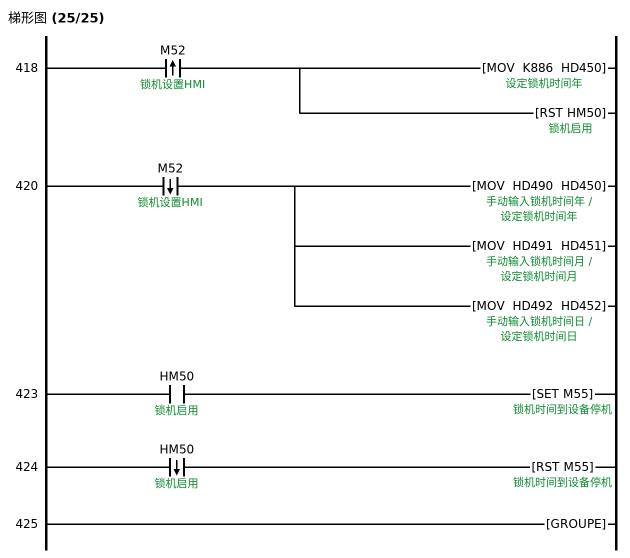
[picture p24: 梯形图 rows 418-425]
LDP    M52	; 锁机设置HMI
MOV    K886 HD450	; 设定锁机时间年
RST    HM50	; 锁机启用
LDF    M52	; 锁机设置HMI
MOV    HD490 HD450	; 手动输入锁机时间年 / 设定锁机时间年
MOV    HD491 HD451	; 手动输入锁机时间月 / 设定锁机时间月
MOV    HD492 HD452	; 手动输入锁机时间日 / 设定锁机时间日
LD     HM50	; 锁机启用
SET    M55	; 锁机时间到设备停机
LDF    HM50	; 锁机启用
RST    M55	; 锁机时间到设备停机
GROUPE

COMMENTS (devices not used above)
M3	急停HMI
M5	NG清料HMI
M6	轴复位HMI
M8	参数默认HMI
M9	产量清零HMI
M10	当前产量清零HMI
M21	軸总復位中
M22	设备复位中
M25	设备清料完成
M2042	轴2_JOG快慢速HMI
M2021	轴1_JOG- HMI
M2022	轴2_JOG- HMI
M2041	轴1_JOG快慢速HMI
M2002	轴2_JOG+ HMI
M1821	与读码器通信异常
D2100	轴1_JOG快速度
D2102	轴1_JOG慢速度
D2104	轴1_JOG速度寄存
D2106	轴1_JOG增量
D2108	轴1_JOG位置寄存
D2110	轴1_回零速度
D2112	轴1_运行速度
D2114	轴1_自动加速度
D2115	轴1_自动减速度
D2116	轴1_JOG加速度
D2117	轴1_JOG减速度
D2118	轴1_定位位置寄存
M2141	轴1_伺服回零中
M1200	快慢速切换HMI
M1020	从1#Y0 左侧三色灯（红）       HMI
HD8	切鼻梁个数计数
HD12	滚刀切料个数计数
M2001	轴1_JOG+ HMI
HD40	Y0当前脉冲值记忆
HD42	Y1当前脉冲值记忆
T2	超声波休眠延时
HD2	超声波休眠时间
T3	超声运行延时
D110	从5读码寄存
D112	从6读码寄存
D114	从7读码寄存
D116	从8读码寄存
D118	从9读码寄存
D120	从10读码寄存
D122	从11读码寄存
D124	从12读码寄存
D126	从13读码寄存
D142	输出脉冲频率浮点数
HD32	生产效率寄存2
HD20	设定产量HMI
HD22	实际产量(切鼻梁个数计数)
HD30	生产效率寄存1
M1600	产量达成
HM30	内置鼻梁标志/外置鼻梁HMI
HD24	滚刀切料个数计数
HD34	生产效率
HM32	校准完成
HM3	急停后切断鼻梁
M18	手动操作记忆标志
HD507	当日实际产量
HD453	设定锁机时间时
HD481	校正时间月
HD482	校正时间日
HD483	校正时间时
D72	年+月+日+时除当前日期得商
HD28	累计产量
X10000	书本到位感应器1（电机侧斜面）       书本到位感应器1
X10001	书本到位感应器2（斜面）             书本到位感应器2
X10002	书本到位感应器3（斜面）             书本到位感应器3
X10003	小车感应光栅
X10004	小车到位感应（对射）
X10005	防压手感应器
X10006	书枰感应器7
X10007	书本感应器8
M2101	轴1_伺服回零HMI
M2102	轴2_伺服回零HMI
M2121	轴1_伺服回零允许
M2122	轴2_伺服回零允许
M2142	轴2_伺服回零中
M2161	轴1_原点确定
M2162	轴2_原点确定
M2181	轴1_定位允许
M2182	轴2_定位允许
M2201	轴1_JOG连续/增量HMI
M2202	轴2_JOG连续/增量HMI
M2241	轴1_增量JOG运行
M2242	轴2_增量JOG运行
M2310	轴1-伺服原点运行HMI
M2311	轴1-伺服定位运行HMI
M2320	轴2-伺服原点运行HMI
M2321	轴2-伺服定位运行HMI
M2510	轴1-伺服原点运行
M2511	轴1-伺服定位运行
M2520	轴2-伺服原点运行
M2521	轴2-伺服定位运行
M2710	轴1-伺服原点位置
M2711	轴1-伺服定位位置
M2720	轴2-伺服原点位置
M2721	轴2-伺服定位位置
HD832	从5，左侧箱号
HD834	从5，右侧箱号
HD836	从5，出料箱号
HD840	从6，左侧箱号
HD842	从6，右侧箱号
HD844	从6，出料箱号
HD848	从7，左侧箱号
HD850	从7，右侧箱号
HD852	从7，出料箱号
HD856	从8，左侧箱号
HD812	从2，出料箱号
HD804	从1，出料箱号
HD868	从9，出料箱号
HD872	从10，左侧箱号
HD874	从10，右侧箱号
HD876	从10，出料箱号
HD880	从11，左侧箱号
HD882	从11，右侧箱号
HD884	从11，出料箱号
HD888	从12，左侧箱号
HD890	从12，右侧箱号
HD892	从12，出料箱号
HD858	从8，右侧箱号
HD860	从8，出料箱号
HD864	从9，左侧箱号
HD866	从9，右侧箱号
D851	轴1-回原点流程
HD828	从4，出料箱号
T422	轴1 启动
M1021	从1#Y1 左侧三色灯（绿）       HMI
D852	轴2-回原流程
T424	轴2定位允许
M1822	主站出料异常
M2312	还书位置运行-HMI
M2512	轴1-还书位置运行
M2712	轴1-还书位置
D810	从站10操作流程
D2501	书本识别启动PLC写1，收到完成信号后PLC置0
D2502	PLC写1，书满暂停，处理完后PLC置0
M1022	从1#Y2 左侧三色灯（黄）       HMI
M1023	从1#Y3 右侧三色灯（红）       HMI
M1024	从1#Y4 右侧三色灯（绿）       HMI
M1025	从1#Y5 右侧三色灯（黄）       HMI
M1026	从1#Y6 出料三色灯（红）       HMI
M1027	从1#Y7 出料三色灯（绿）       HMI
M1028	从1#Y10 出料三色灯（黄）       HMI
M1030	从1#Y12 进料输送皮带（正常）       HMI
M1040	从2#Y0 左侧三色灯（红）       HMI
M1041	从2#Y1 左侧三色灯（绿）       HMI
M1042	从2#Y2 左侧三色灯（黄）       HMI
M1043	从2#Y3 右侧三色灯（红）       HMI
M1044	从2#Y4 右侧三色灯（绿）       HMI
M1045	从2#Y5 右侧三色灯（黄）       HMI
M1046	从2#Y6 出料三色灯（红）       HMI
M1047	从2#Y7 出料三色灯（绿）       HMI
M1048	从2#Y10 出料三色灯（黄）       HMI
M1050	从2#Y12 进料输送皮带（正常）       HMI
M1060	从3#Y0 左侧三色灯（红）       HMI
M1061	从3#Y1 左侧三色灯（绿）       HMI
M1062	从3#Y2 左侧三色灯（黄）       HMI
M1063	从3#Y3 右侧三色灯（红）       HMI
M1064	从3#Y4 右侧三色灯（绿）       HMI
M1065	从3#Y5 右侧三色灯（黄）       HMI
M1066	从3#Y6 出料三色灯（红）       HMI
M1067	从3#Y7 出料三色灯（绿）       HMI
M1068	从3#Y10 出料三色灯（黄）       HMI
M1070	从3#Y12 进料输送皮带（正常）       HMI
M4026	从1#Y6 出料三色灯（红）
M4027	从1#Y7 出料三色灯（绿）
M4028	从1#Y10 出料三色灯（黄）
M4066	从2#Y6 出料三色灯（红）
M4067	从2#Y7 出料三色灯（绿）
M4068	从2#Y10 出料三色灯（黄）
M4106	从3#Y6 出料三色灯（红）
M4107	从3#Y7 出料三色灯（绿）
M4108	从3#Y10 出料三色灯（黄）
M103	从站4#进料皮带速度切换=0 正常，=1低速
M104	从站5#进料皮带速度切换=0 正常，=1低速
M105	从站6#进料皮带速度切换=0 正常，=1低速
M106	从站7#进料皮带速度切换=0 正常，=1低速
M107	从站8#进料皮带速度切换=0 正常，=1低速
M108	从站9#进料皮带速度切换=0 正常，=1低速
M109	从站10#进料皮带速度切换=0 正常，=1低速
M110	从站11#进料皮带速度切换=0 正常，=1低速
M111	从站12#进料皮带速度切换=0 正常，=1低速
M112	从站13#进料皮带速度切换=0 正常，=1低速
M1610	主站已进料
T401	主站出料超时
M1611	从1已进料
M132	从5#出料
M133	从5#左出料
M134	从5#右出料
M135	从6#出料
M136	从6#左出料
M137	从6#右出料
M138	从7#出料
M139	从7#左出料
M140	从7#右出料
M141	从8#出料
M142	从8#左出料
M143	从8#右出料
M144	从9#出料
M145	从9#左出料
M146	从9#右出料
M147	从10#出料
M148	从10#左出料
M149	从10#右出料
M150	从11#出料
M151	从11#左出料
M152	从11#右出料
M153	从12#出料
M154	从12#左出料
M155	从12#右出料
M156	从13#出料
M157	从13#左出料
M158	从13#右出料
D804	从站4操作流程
D805	从站5操作流程
D806	从站6操作流程
D807	从站7操作流程
D808	从站8操作流程
D809	从站9操作流程
D811	从站11操作流程
D812	从站12操作流程
D813	从站13操作流程